Universal Robots PolyScope program: New_Poses.urp

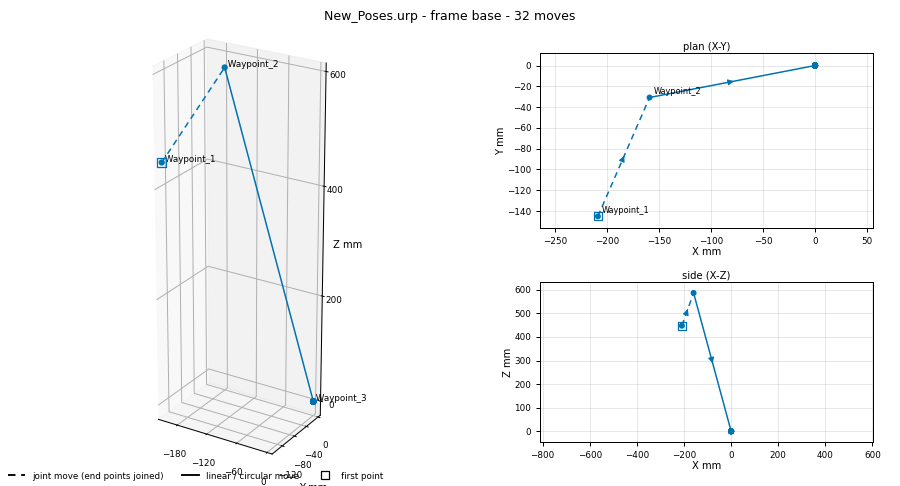
[picture p0: tool path of New_Poses.urp in frame base, 32 of 32 moves have a stored position in this frame; points joined in program order, loops and branches not executed]
Program New_Poses (createdIn=3.15.4.106291 lastSavedIn=3.15.4.106291)
Robot Program (runOnlyOnce=false)
  MoveJ speed 180.02 deg/s, acceleration 719.98 deg/s^2 (useActiveTCP=true)
    Waypoint Waypoint_1: motionParameters(blendRadius=0); TCP in base x=-209.026 y=-145.135 z=447.631 mm, rx=2.1855 ry=-0.0378 rz=2.2231 rad; joints [2.067, -1.08, -72.287, -105.655, 85.984, -90.037] deg
  MoveJ speed 180.02 deg/s, acceleration 719.98 deg/s^2 (useActiveTCP=true)
    Waypoint Waypoint_2: motionParameters(blendRadius=0); TCP in base x=-159.306 y=-30.767 z=586.828 mm, rx=-2.1994 ry=-0.0494 rz=-2.1993 rad; joints [-23.207, -34.238, -51.481, -94.284, 115.743, -90.039] deg
  MoveL speed 1000 mm/s, acceleration 4000 mm/s^2 (useActiveTCP=true)
    Waypoint Waypoint_3: motionParameters(blendRadius=0); TCP in base x=0 y=0 z=0 mm, rx=0 ry=0 rz=0 rad; joints [-70.784, -43.562, 0, -136.53, 115.284, -89.849] deg
  MoveL speed 1000 mm/s, acceleration 4000 mm/s^2 (useActiveTCP=true)
    Waypoint Waypoint_4: motionParameters(blendRadius=0); TCP in base x=0 y=0 z=0 mm, rx=0 ry=0 rz=0 rad; joints [-80.69, -38.593, 0, -141.508, 125.19, -89.867] deg
  MoveL speed 1000 mm/s, acceleration 4000 mm/s^2 (useActiveTCP=true)
    Waypoint Waypoint_5: motionParameters(blendRadius=0); TCP in base x=0 y=0 z=0 mm, rx=0 ry=0 rz=0 rad; joints [-125.657, -38.582, 0, -141.518, 125.158, -89.867] deg
  MoveL speed 1000 mm/s, acceleration 4000 mm/s^2 (useActiveTCP=true)
    Waypoint Waypoint_6: motionParameters(blendRadius=0); TCP in base x=0 y=0 z=0 mm, rx=0 ry=0 rz=0 rad; joints [-170.627, -38.586, 0, -141.515, 125.127, -89.867] deg
  MoveL speed 1000 mm/s, acceleration 4000 mm/s^2 (useActiveTCP=true)
    Waypoint Waypoint_7: motionParameters(blendRadius=0); TCP in base x=0 y=0 z=0 mm, rx=0 ry=0 rz=0 rad; joints [-184.796, -38.072, 0, -141.81, 139.297, -89.718] deg
  MoveL speed 1000 mm/s, acceleration 4000 mm/s^2 (useActiveTCP=true)
    Waypoint Waypoint_8: motionParameters(blendRadius=0); TCP in base x=0 y=0 z=0 mm, rx=0 ry=0 rz=0 rad; joints [-211.327, -46.976, 0, -140.802, 123.743, -59.495] deg
  MoveL speed 1000 mm/s, acceleration 4000 mm/s^2 (useActiveTCP=true)
    Waypoint Waypoint_9: motionParameters(blendRadius=0); TCP in base x=0 y=0 z=0 mm, rx=0 ry=0 rz=0 rad; joints [-168.012, -40.025, 0, -132.847, 123.446, -56.76] deg
  MoveL speed 1000 mm/s, acceleration 4000 mm/s^2 (useActiveTCP=true)
    Waypoint Waypoint_10: motionParameters(blendRadius=0); TCP in base x=0 y=0 z=0 mm, rx=0 ry=0 rz=0 rad; joints [-124.595, -35.179, 0, -131.412, 124.384, -65.773] deg
  MoveL speed 1000 mm/s, acceleration 4000 mm/s^2 (useActiveTCP=true)
    Waypoint Waypoint_11: motionParameters(blendRadius=0); TCP in base x=0 y=0 z=0 mm, rx=0 ry=0 rz=0 rad; joints [-79.921, -35.17, 0, -137.84, 125.104, -82.046] deg
  MoveL speed 1000 mm/s, acceleration 4000 mm/s^2 (useActiveTCP=true)
    Waypoint Waypoint_12: motionParameters(blendRadius=0); TCP in base x=0 y=0 z=0 mm, rx=0 ry=0 rz=0 rad; joints [-35.048, -36.441, 0, -135.197, 125.415, -86.418] deg
  MoveL speed 1000 mm/s, acceleration 4000 mm/s^2 (useActiveTCP=true)
    Waypoint Waypoint_13: motionParameters(blendRadius=0); TCP in base x=0 y=0 z=0 mm, rx=0 ry=0 rz=0 rad; joints [-33.112, -34.566, 0, -129.508, 126.09, -83.492] deg
  MoveL speed 1000 mm/s, acceleration 4000 mm/s^2 (useActiveTCP=true)
    Waypoint Waypoint_14: motionParameters(blendRadius=0); TCP in base x=0 y=0 z=0 mm, rx=0 ry=0 rz=0 rad; joints [-78.129, 12.719, -82.828, -63.81, 121.654, -56.47] deg
  MoveL speed 1000 mm/s, acceleration 4000 mm/s^2 (useActiveTCP=true)
    Waypoint Waypoint_15: motionParameters(blendRadius=0); TCP in base x=0 y=0 z=0 mm, rx=0 ry=0 rz=0 rad; joints [-131.323, 15.452, -89.66, -51.719, 112.223, -24.632] deg
  MoveL speed 1000 mm/s, acceleration 4000 mm/s^2 (useActiveTCP=true)
    Waypoint Waypoint_16: motionParameters(blendRadius=0); TCP in base x=0 y=0 z=0 mm, rx=0 ry=0 rz=0 rad; joints [-173.74, -24.469, -21.076, -99.143, 107.545, -11.709] deg
  MoveL speed 1000 mm/s, acceleration 4000 mm/s^2 (useActiveTCP=true)
    Waypoint Waypoint_17: motionParameters(blendRadius=0); TCP in base x=0 y=0 z=0 mm, rx=0 ry=0 rz=0 rad; joints [-198.556, -52.22, 0, -137.664, 118.881, -24.691] deg
  MoveL speed 1000 mm/s, acceleration 4000 mm/s^2 (useActiveTCP=true)
    Waypoint Waypoint_18: motionParameters(blendRadius=0); TCP in base x=0 y=0 z=0 mm, rx=0 ry=0 rz=0 rad; joints [-215.61, -38.292, 0, -143.062, 125.077, -93.519] deg
  MoveL speed 1000 mm/s, acceleration 4000 mm/s^2 (useActiveTCP=true)
    Waypoint Waypoint_19: motionParameters(blendRadius=0); TCP in base x=0 y=0 z=0 mm, rx=0 ry=0 rz=0 rad; joints [-260.626, -38.31, 0, -143.044, 125.093, -93.519] deg
  MoveL speed 1000 mm/s, acceleration 4000 mm/s^2 (useActiveTCP=true)
    Waypoint Waypoint_20: motionParameters(blendRadius=0); TCP in base x=0 y=0 z=0 mm, rx=0 ry=0 rz=0 rad; joints [-305.66, -38.32, 0, -143.034, 125.127, -93.52] deg
  MoveL speed 1000 mm/s, acceleration 4000 mm/s^2 (useActiveTCP=true)
    Waypoint Waypoint_21: motionParameters(blendRadius=0); TCP in base x=0 y=0 z=0 mm, rx=0 ry=0 rz=0 rad; joints [-350.693, -38.317, 0, -143.038, 125.159, -93.521] deg
  MoveL speed 1000 mm/s, acceleration 4000 mm/s^2 (useActiveTCP=true)
    Waypoint Waypoint_22: motionParameters(blendRadius=0); TCP in base x=0 y=0 z=0 mm, rx=0 ry=0 rz=0 rad; joints [-395.685, -37.678, 0, -140.911, 125.205, -91.907] deg
  MoveL speed 1000 mm/s, acceleration 4000 mm/s^2 (useActiveTCP=true)
    Waypoint Waypoint_23: motionParameters(blendRadius=0); TCP in base x=0 y=0 z=0 mm, rx=0 ry=0 rz=0 rad; joints [-365.672, -35.911, 0, -135.386, 138.952, -87.433] deg
  MoveL speed 1000 mm/s, acceleration 4000 mm/s^2 (useActiveTCP=true)
    Waypoint Waypoint_24: motionParameters(blendRadius=0); TCP in base x=0 y=0 z=0 mm, rx=0 ry=0 rz=0 rad; joints [-352.166, -33.422, 0, -139.562, 125.571, -89.923] deg
  MoveL speed 1000 mm/s, acceleration 4000 mm/s^2 (useActiveTCP=true)
    Waypoint Waypoint_25: motionParameters(blendRadius=0); TCP in base x=0 y=0 z=0 mm, rx=0 ry=0 rz=0 rad; joints [-307.407, -13.413, -31.186, -121.619, 125.085, -98.539] deg
  MoveL speed 1000 mm/s, acceleration 4000 mm/s^2 (useActiveTCP=true)
    Waypoint Waypoint_26: motionParameters(blendRadius=0); TCP in base x=0 y=0 z=0 mm, rx=0 ry=0 rz=0 rad; joints [-259.954, -20.834, -15.077, -136.482, 123.168, -115.217] deg
  MoveL speed 1000 mm/s, acceleration 4000 mm/s^2 (useActiveTCP=true)
    Waypoint Waypoint_27: motionParameters(blendRadius=0); TCP in base x=0 y=0 z=0 mm, rx=0 ry=0 rz=0 rad; joints [-247.101, 4.002, -79.408, -83.287, 114.216, -111.357] deg
  MoveL speed 1000 mm/s, acceleration 4000 mm/s^2 (useActiveTCP=true)
    Waypoint Waypoint_28: motionParameters(blendRadius=0); TCP in base x=0 y=0 z=0 mm, rx=0 ry=0 rz=0 rad; joints [-212.474, -31.224, 0, -149.484, 121.382, -129.167] deg
  MoveL speed 1000 mm/s, acceleration 4000 mm/s^2 (useActiveTCP=true)
    Waypoint Waypoint_29: motionParameters(blendRadius=0); TCP in base x=0 y=0 z=0 mm, rx=0 ry=0 rz=0 rad; joints [-258.595, 18.77, -84.433, -84.928, 124.763, -101.725] deg
  MoveL speed 1000 mm/s, acceleration 4000 mm/s^2 (useActiveTCP=true)
    Waypoint Waypoint_30: motionParameters(blendRadius=0); TCP in base x=0 y=0 z=0 mm, rx=0 ry=0 rz=0 rad; joints [-313.311, 21.13, -93.311, -64.359, 123.785, -64.631] deg
  MoveL speed 1000 mm/s, acceleration 4000 mm/s^2 (useActiveTCP=true)
    Waypoint Waypoint_31: motionParameters(blendRadius=0); TCP in base x=0 y=0 z=0 mm, rx=0 ry=0 rz=0 rad; joints [-355.87, -19.385, -27.228, -105.67, 121.693, -50.19] deg
  MoveL speed 1000 mm/s, acceleration 4000 mm/s^2 (useActiveTCP=true)
    Waypoint Waypoint_32: motionParameters(blendRadius=0); TCP in base x=0 y=0 z=0 mm, rx=0 ry=0 rz=0 rad; joints [-393.404, -44.672, 0, -134.53, 122.328, -56.348] deg
